// TIA Portal project "Counter Timer Uygulama" (V17)

(* hardware
DEVICE "S71500/ET200MP-Station_1"  S7-1500 station
   slot 0: "Profilschiene_0"  6ES7 590-1***0-0AA0
   slot 1: "PLC_1"  CPU 1511-1 PN  6ES7 511-1AK00-0AB0  V1.8
   slot 2: "AI 8xU/I/RTD/TC ST_1"  AI 8xU/I/RTD/TC ST  6ES7 531-7KF00-0AB0  V2.0
   slot 3: "AI 8xU/I/RTD/TC ST_2"  AI 8xU/I/RTD/TC ST  6ES7 531-7KF00-0AB0  V2.0
   slot 4: "AI 8xU/I/RTD/TC ST_3"  AI 8xU/I/RTD/TC ST  6ES7 531-7KF00-0AB0  V2.0
   slot 5: "AI 8xU/I/RTD/TC ST_4"  AI 8xU/I/RTD/TC ST  6ES7 531-7KF00-0AB0  V2.0
   slot 6: "DI 16x24VDC BA_1"  DI 16x24VDC BA  6ES7 521-1BH10-0AA0  V1.0
*)

// ===== PLC "PLC_1"  CPU 1511-1 PN =====

VAR_GLOBAL   // PLC tag table "Standard-Variablentabelle"
   "START" AT %E0.0 : Bool;
   "MOTOR" AT %A0.0 : Bool;
   "STOP" AT %E0.1 : Bool;
   "Tag_1" AT %M0.0 : Bool;
   "Sensör A" AT %I0.2 : Bool;
   "Tag_2" AT %Q0.1 : Bool;
   "Tag_3" AT %M100.0 : Bool;
   "Tag_4" AT %M0.1 : Bool;
   "Tag_5" AT %M0.2 : Bool;
   "Sensör B" AT %I0.3 : Bool;
   "Tag_7" AT %M100.1 : Bool;
   "Tag_6" AT %MW100 : Int;
   "Tag_8" AT %M0.4 : Bool;
   "Tag_9" AT %QD30 : DWord;
   "Tag_10" AT %MD100 : Time;
   "Tag_11" AT %MD150 : DInt;
   "Tag_12" AT %QD34 : DInt;
END_VAR

// folder: System blocks/Program resources

DATA_BLOCK "IEC_Timer_0_DB"   // DB1
{ S7_Optimized_Access := 'TRUE' }
AUTHOR : Simatic
FAMILY : IEC
NAME : IEC_TMR
VERSION : 1.0
// stored: InstanceOfName IEC_TIMER
"IEC_TIMER"
BEGIN
END_DATA_BLOCK

DATA_BLOCK "IEC_Counter_0_DB"   // DB2
{ S7_Optimized_Access := 'TRUE' }
AUTHOR : Simatic
FAMILY : IEC
NAME : CNTR
VERSION : 1.0
// stored: InstanceOfName IEC_COUNTER
"IEC_COUNTER"
BEGIN
END_DATA_BLOCK

// folder: (top level)

FUNCTION "MHJ-PLC-Lab-Function-S71500" : Void   // FC9000, SCL
{ S7_Optimized_Access := 'TRUE' }
VERSION : 0.1
   VAR_TEMP
      Value : Byte;
      ForCounter : Int;
   END_VAR
   VAR CONSTANT
      Value_01_DW : DWord := 16#1223_5486;
      Value_02_DW : DWord := 16#A6C9_D1F5;
   END_VAR
BEGIN

   #Value:=PEEK(area := 16#82,
        dbNumber := 0,
        byteOffset := 511);
   #Value := #Value + 1;

   POKE(area := 16#82,
        dbNumber := 0,
        byteOffset := 511,
        value := #Value);

   POKE(area := 16#82,
        dbNumber := 0,
        byteOffset := 1016,
        value := #Value_01_DW);
   POKE(area := 16#82,
        dbNumber := 0,
        byteOffset := 1020,
        value := #Value_02_DW);

   FOR #ForCounter := 0 TO 63 DO
       #Value:=PEEK(area := 16#1,
            dbNumber := 0,
            byteOffset := #ForCounter);
       POKE(area := 16#81,
            dbNumber := 0,
            byteOffset := #ForCounter,
            value := #Value);
   END_FOR;
   #Value := PEEK(area := 16#1,
                  dbNumber := 0,
                  byteOffset := 512);
   POKE(area := 16#82,
        dbNumber := 0,
        byteOffset := 512,
        value := #Value);
END_FUNCTION

ORGANIZATION_BLOCK "Main"   // OB1, LAD, ProgramCycle
TITLE = "Main Program Sweep (Cycle)"
{ S7_Optimized_Access := 'TRUE' }
VERSION : 0.1
   VAR_INPUT
      Initial_Call : Bool;   // Initial call of this OB
      Remanence : Bool;   // =True, if remanent data are available
   END_VAR
   VAR_TEMP   // added for the SCL form of the ladder/FBD networks
      _w1 : Bool;
   END_VAR
BEGIN

REGION Network 1
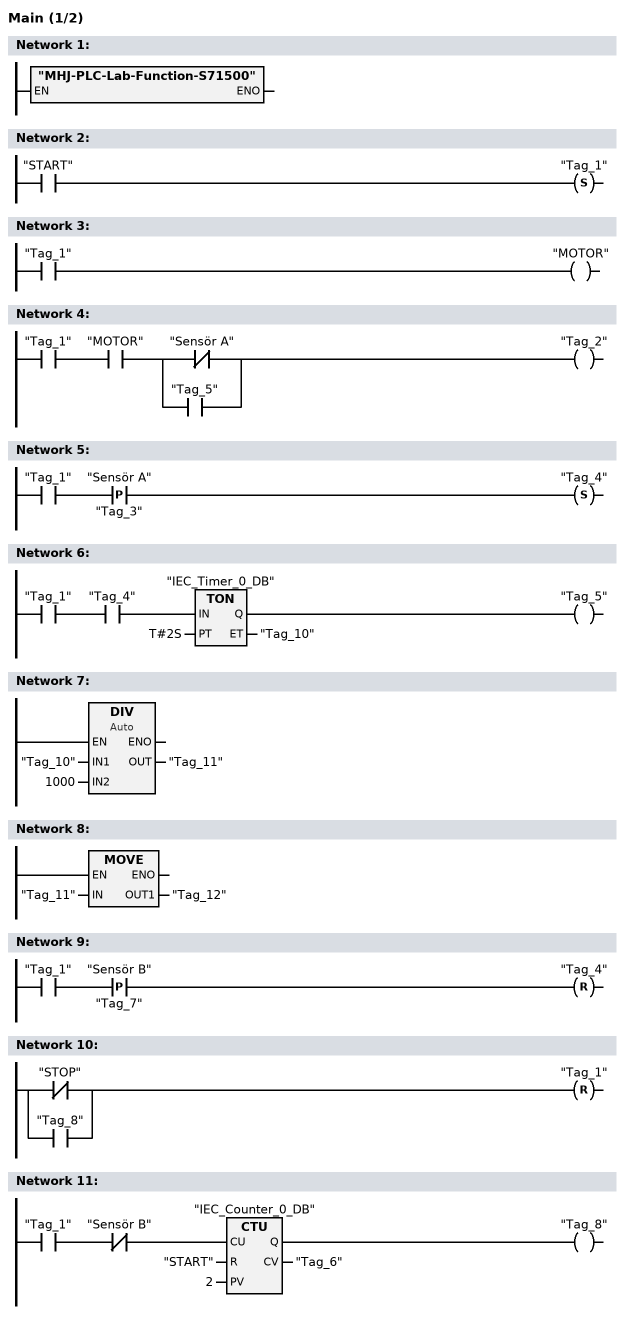
   RUNG wire#powerrail
      "MHJ-PLC-Lab-Function-S71500"()
   END_RUNG
   // the same network as SCL:
   "MHJ-PLC-Lab-Function-S71500"();
END_REGION

REGION Network 2
   RUNG wire#powerrail
      Contact( "START" )
      S_Coil( "Tag_1" )
   END_RUNG
   // the same network as SCL:
   IF "START" THEN "Tag_1" := TRUE; END_IF;
END_REGION

REGION Network 3
   RUNG wire#powerrail
      Contact( "Tag_1" )
      Coil( "MOTOR" )
   END_RUNG
   // the same network as SCL:
   "MOTOR" := "Tag_1";
END_REGION

REGION Network 4
   RUNG wire#powerrail
      Contact( "Tag_1" )
      Contact( "MOTOR" )
      wire#w1
      I_Contact( "Sensör A" )
      wire#w2
      Coil( "Tag_2" )
   END_RUNG
   RUNG wire#w1
      Contact( "Tag_5" )
   END_RUNG wire#w2
   // the same network as SCL:
   "Tag_2" := "Tag_1" AND "MOTOR" AND (NOT "Sensör A" OR "Tag_5");
END_REGION

REGION Network 5
   RUNG wire#powerrail
      Contact( "Tag_1" )
      P_Contact(operand := "Sensör A", bit := "Tag_3")
      S_Coil( "Tag_4" )
   END_RUNG
   // the same network as SCL:
   #_w1 := "Tag_1" AND "Sensör A" AND NOT "Tag_3";   // rising edge of "Sensör A"
   "Tag_3" := "Sensör A";
   IF #_w1 THEN "Tag_4" := TRUE; END_IF;
END_REGION

REGION Network 6
   "IEC_Timer_0_DB".TON(IN := "Tag_1" AND "Tag_4", PT := T#2S, ET => "Tag_10");
   "Tag_5" := "IEC_Timer_0_DB".Q;
END_REGION

REGION Network 7
   RUNG wire#powerrail
      Div(in1 := "Tag_10", in2 := 1000, out => "Tag_11")
   END_RUNG
   // the same network as SCL:
   "Tag_11" := "Tag_10" / 1000;
END_REGION

REGION Network 8
   RUNG wire#powerrail
      Move(in := "Tag_11", out1 => "Tag_12")
   END_RUNG
   // the same network as SCL:
   "Tag_12" := "Tag_11";
END_REGION

REGION Network 9
   RUNG wire#powerrail
      Contact( "Tag_1" )
      P_Contact(operand := "Sensör B", bit := "Tag_7")
      R_Coil( "Tag_4" )
   END_RUNG
   // the same network as SCL:
   #_w1 := "Tag_1" AND "Sensör B" AND NOT "Tag_7";   // rising edge of "Sensör B"
   "Tag_7" := "Sensör B";
   IF #_w1 THEN "Tag_4" := FALSE; END_IF;
END_REGION

REGION Network 10
   RUNG wire#powerrail
      I_Contact( "STOP" )
      wire#w1
      R_Coil( "Tag_1" )
   END_RUNG
   RUNG wire#powerrail
      Contact( "Tag_8" )
   END_RUNG wire#w1
   // the same network as SCL:
   IF NOT "STOP" OR "Tag_8" THEN "Tag_1" := FALSE; END_IF;
END_REGION

REGION Network 11
   "IEC_Counter_0_DB".CTU(CU := "Tag_1" AND NOT "Sensör B", R := "START", PV := 2, CV => "Tag_6");
   "Tag_8" := "IEC_Counter_0_DB".Q;
END_REGION

REGION Network 12
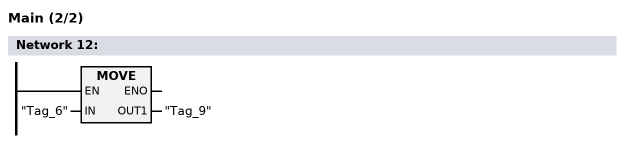
   RUNG wire#powerrail
      Move(in := "Tag_6", out1 => "Tag_9")
   END_RUNG
   // the same network as SCL:
   "Tag_9" := "Tag_6";
END_REGION
END_ORGANIZATION_BLOCK